(* LS Electric XG5000 project: TK-2026-XEC *)
(* PLC LSPLC *)

PROGRAM NewProgram (* task: 스캔 프로그램 *)
// ===============================================================
//  본문 로직
// ===============================================================

// [STEP 0] 펄스 및 운전 모드 판정
trig_RemotePump(CLK := xRemote_PumpStart, Q => xRemotePumpPulse);
trig_RemoteDrain(CLK := xRemote_DrainStart, Q => xRemoteDrainPulse);
trig_AlarmReset(CLK := xAlarmReset_PB OR xRemote_AlarmReset, Q => xAlarmResetPulse);
trig_CommHeartbeat(CLK := xComm_Heartbeat, Q => xCommHeartbeatPulse);

xIsAutoMode := xManualMode_SW;

// [STEP 1] 아날로그 입력 스케일링
rDiffPressure := INT_TO_REAL(iRaw_DiffPressure) * 300.0 / 27648.0;
rTDS_Value    := INT_TO_REAL(iRaw_TDS) * 10000.0 / 27648.0;
rHumidity_S1  := INT_TO_REAL(iRaw_Humidity_S1) * 100.0 / 27648.0;
rHumidity_S2  := INT_TO_REAL(iRaw_Humidity_S2) * 100.0 / 27648.0;
rSumpTemp     := (INT_TO_REAL(iRaw_SumpTemp) * 100.0 / 27648.0) - 20.0;
rAmbientTemp  := (INT_TO_REAL(iRaw_AmbientTemp) * 100.0 / 27648.0) - 20.0;

// [STEP 2] 센서 Fail-safe 검증
xSensorFault_DP   := (iRaw_DiffPressure <= 0) OR (rDiffPressure > 310.0);
xSensorFault_TDS  := (iRaw_TDS <= 0) OR (rTDS_Value > 10200.0);
xSensorFault_Hum  := (rHumidity_S1 < 0.0) OR (rHumidity_S1 > 101.0)
                  OR (rHumidity_S2 < 0.0) OR (rHumidity_S2 > 101.0);
xSensorFault_Temp := (rSumpTemp < -25.0) OR (rSumpTemp > 90.0);

xAlarm_SensorFault := xSensorFault_DP OR xSensorFault_TDS OR xSensorFault_Hum OR xSensorFault_Temp;

// [STEP 3] EBCT 실시간 모니터링
IF (rDesignFlow_CMM > 0.0) AND (rDesignArea_m2 > 0.0) THEN
    rEBCT_Check := H_TOTAL_MEDIA_M / ((rDesignFlow_CMM / 60.0) / rDesignArea_m2);
ELSE
    rEBCT_Check := 0.0;
END_IF;

// [STEP 4] 차압 관리
rDP_Trend_RateOfRise := (rDiffPressure - rDP_Trend_Prev) * 3600.0;
rDP_Trend_Prev := rDiffPressure;
xAlarm_pHBreakthrough := (rDP_Trend_RateOfRise > DP_RATE_ALARM_MMH) AND NOT xSensorFault_DP;

xAlarm_DP_Backwash := (rDiffPressure >= DP_BACKWASH_TRIGGER)
                   AND (rDiffPressure < DP_SHUTDOWN)
                   AND NOT xSensorFault_DP;
xValveBackwash := xAlarm_DP_Backwash AND xIsAutoMode;

IF xAlarmResetPulse THEN
    xAlarm_DP_High := FALSE;
ELSIF (rDiffPressure >= DP_SHUTDOWN) AND NOT xSensorFault_DP THEN
    xAlarm_DP_High := TRUE;
END_IF;

// [STEP 5] 송풍기 제어
IF xAlarm_DP_High OR xAlarm_SensorFault THEN
    xBlowerRun := FALSE;
ELSIF xIsAutoMode THEN
    xBlowerRun := TRUE;
ELSE
    xBlowerRun := FALSE;
END_IF;

// [STEP 6] 살수펌프 제어
ton_PumpMinRun(IN := xPumpRun, PT := PUMP_MIN_RUN_SEC, Q => xPumpMinDone);
ton_PumpMaxRun(IN := xPumpRun, PT := PUMP_MAX_RUN_SEC, Q => xPumpMaxDone);

xAlarm_PumpOverrun := xPumpMaxDone;

IF xIsAutoMode AND NOT xAlarm_SensorFault THEN
    IF (rHumidity_S1 < HUMID_LOW_SETPOINT) OR (rHumidity_S2 < HUMID_LOW_SETPOINT) THEN
        xPumpRun := TRUE;
    ELSIF (rHumidity_S1 >= HUMID_HIGH_SETPOINT)
       AND (rHumidity_S2 >= HUMID_HIGH_SETPOINT)
       AND xPumpMinDone THEN
        xPumpRun := FALSE;
    END_IF;

    IF xAlarm_PumpOverrun THEN
        xPumpRun := FALSE;
    END_IF;
ELSE
    xPumpRun := FALSE;
END_IF;

// [STEP 7] 동파방지 히터 제어
ton_HeaterMinOff(IN := NOT xHeaterRun, PT := HEATER_MIN_OFF_SEC, Q => xHeaterMinOffDone);

xAlarm_HeaterFault := (rSumpTemp >= HEATER_FAULT_TEMP) AND NOT xSensorFault_Temp;

IF xAlarm_HeaterFault OR xSensorFault_Temp THEN
    xHeaterRun := FALSE;
ELSIF (rSumpTemp <= HEATER_ON_TEMP) OR (rAmbientTemp <= AMBIENT_PREHEAT_TEMP) THEN
    IF xHeaterMinOffDone THEN
        xHeaterRun := TRUE;
    END_IF;
ELSIF rSumpTemp >= HEATER_OFF_TEMP THEN
    xHeaterRun := FALSE;
END_IF;

// [STEP 8] TDS 드레인 시퀀스
ton_DrainSequence(IN := (iDrainSeqState = 1) AND (rTDS_Value < TDS_DRAIN_STOP), PT := DRAIN_SEQ_DELAY, Q => xDrainDelayDone);

CASE iDrainSeqState OF
    0:
        xValveDrain  := FALSE;
        xValveMakeup := FALSE;
        IF (rTDS_Value >= TDS_DRAIN_START) AND NOT xSensorFault_TDS AND xIsAutoMode THEN
            iDrainSeqState := 1;
        END_IF;

    1:
        xValveDrain  := TRUE;
        xValveMakeup := FALSE;
        IF xDrainDelayDone THEN
            iDrainSeqState := 2;
        END_IF;
        IF xSumpLevel_Low THEN
            iDrainSeqState := 0;
            xAlarm_SumpLow := TRUE;
        END_IF;

    2:
        xValveDrain  := FALSE;
        xValveMakeup := TRUE;
        IF xSumpLevel_High THEN
            iDrainSeqState := 3;
        END_IF;

    3:
        xValveDrain  := FALSE;
        xValveMakeup := FALSE;
        iDrainSeqState := 0;

    ELSE
        iDrainSeqState := 0;
END_CASE;

xAlarm_SumpLow := xSumpLevel_Low;

// [STEP 9] SCADA 통신 워치독
ton_CommWatchdog(IN := NOT xCommHeartbeatPulse, PT := COMM_WATCHDOG_T, Q => xCommWatchdogDone);

IF xCommWatchdogDone THEN
    xAlarm_CommLost := TRUE;
    xRemoteModeActive := FALSE;
ELSE
    xAlarm_CommLost := FALSE;
    xRemoteModeActive := xRemoteMode_Cmd;
END_IF;

// [STEP 10] 원격 명령 처리
IF xRemoteModeActive THEN
    IF xRemotePumpPulse THEN
        xPumpRun := TRUE;
    END_IF;

    IF xRemoteDrainPulse AND (iDrainSeqState = 0) THEN
        iDrainSeqState := 1;
    END_IF;
END_IF;

END_FUNCTION_BLOCK
END_PROGRAM